(* PLC project , Siemens AG TIA Portal V17 *)

PROGRAM MainOb1

PROGRAM MainOb1
VAR
    Run : BOOL := TRUE;
END_VAR
END_PROGRAM
END_PROGRAM

PROGRAM DiagFc

FUNCTION DiagFc : INT
DiagFc := 7;
END_FUNCTION
END_PROGRAM

PROGRAM LegacyDb

DATA_BLOCK LegacyDb
END_DATA_BLOCK
END_PROGRAM
